// TIA Portal V19 export
FUNCTION "Lamp" : Bool   // FC145, LAD
// stored: Access Published, SetENOAutomatically false
   VAR_INPUT
      Signal : Bool;
   END_VAR
BEGIN

REGION Network 1
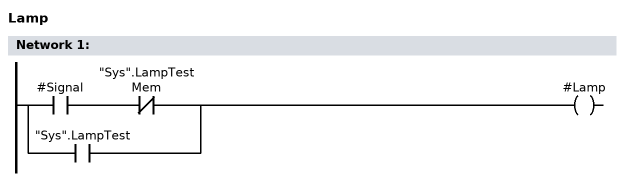
   RUNG wire#powerrail
      Contact( #Signal )
      I_Contact( "Sys".LampTestMem )
      wire#w1
      Coil( #Lamp )
   END_RUNG
   RUNG wire#powerrail
      Contact( "Sys".LampTest )
   END_RUNG wire#w1
   // the same network as SCL:
   #Lamp := (#Signal AND NOT "Sys".LampTestMem) OR "Sys".LampTest;
END_REGION
END_FUNCTION
